{attribute 'qualified_only'}
{attribute 'strict'}
{attribute 'conditionalshow'}
TYPE E_SimMovitracState :
(
	ControllerInhibit := 1,
	RapidStop := 2,
	Halt := 3,
	HoldControl := 4,
	Enable := 5
);
END_TYPE

(* stored: Version 1.1.0.1, ProductVersion 3.1.4024.12
   DUT E_SimMovitracState: Id {4162896b-2c36-0c79-0e5b-2c9cdc67bec2} *)
